// TwinCAT 3 PLC project Test_Conexion
// ProgramVersion: 3.1.4024.0
// libraries:
//   Tc2_Standard, * (Beckhoff Automation GmbH)
//   Tc2_System, * (Beckhoff Automation GmbH)
//   Tc3_Module, * (Beckhoff Automation GmbH)
// project tree:
//   GVLs/ GVL_FMS201.TcGVL, GVL_ILUMINACION.TcGVL
//   / PlcTask.TcTTO
//   POUs/ MAIN.TcPOU
// real-time tasks:
//   TASK PlcTask: cycle T#10ms, priority 20, ADS port 350

CONFIGURATION Test_Conexion
    RESOURCE PLC ON TwinCAT3
        TASK PlcTask(INTERVAL := T#10ms, PRIORITY := 20);
        PROGRAM MAIN WITH PlcTask : MAIN;
    END_RESOURCE
END_CONFIGURATION

// ---- GVLs/GVL_FMS201.TcGVL
{attribute 'qualified_only'}
VAR_GLOBAL
	bTrigger        : BOOL;
    bInspeccionando : BOOL;
    iResultado      : INT;
    sResultado      : STRING(80);
    bResultadoListo : BOOL;
END_VAR

// ---- GVLs/GVL_ILUMINACION.TcGVL
{attribute 'qualified_only'}
VAR_GLOBAL
	bAroLuzOn: BOOL;
	bAroLuzOff: BOOL;
END_VAR

// ---- POUs/MAIN.TcPOU
PROGRAM MAIN
VAR
	bTestSimple: BOOL;
END_VAR

END_PROGRAM
